// TIA Portal V17 export
// export: Created 2023-05-01T07:54:19.7526705Z, ExportSetting WithDefaults, DisplayName Totally Integrated Automation Portal, DisplayVersion V17, DisplayName TIA Portal Openness, DisplayVersion V17, DisplayName TIA Portal Version Control Interface, DisplayVersion V17, DisplayName STEP 7 Professional, DisplayVersion V17, DisplayName STEP 7 Safety, DisplayVersion V17, DisplayName WinCC Advanced / Unified PC, DisplayVersion V17
FUNCTION "FC_NormScaleAnalogInput" : Void   // FC1, LAD
{ S7_Optimized_Access := 'TRUE' }
VERSION : 0.1
// stored: AutoNumber true, IsIECCheckEnabled false, SetENOAutomatically false, UDAEnableTagReadback false
   VAR_INPUT
      AnalogInput : Int;   // Analog input [value 0 - 27648]
      minScaledValue : Real;   // lower value for scaled value Real
      maxScaledValue : Real;   // Upper value for scaled value Real
   END_VAR
   VAR_OUTPUT
      AnalogInputReal : Real;   // Scaled analog value Real
   END_VAR
   VAR_TEMP
      normAnalogValue : Real;
   END_VAR
   VAR CONSTANT
      LOWERINT : Int := 0;
      UPPERINT : Int := 27648;
   END_VAR
BEGIN

REGION Network 1
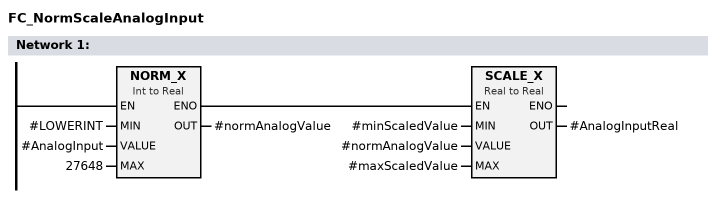
   RUNG wire#powerrail
      { S7_Templates := "[SrcType := Int, DestType := Real]" } Normalize(min := #LOWERINT, value := #AnalogInput, max := 27648, out => #normAnalogValue)
      { S7_Templates := "[SrcType := Real, DestType := Real]" } Scale(min := #minScaledValue, value := #normAnalogValue, max := #maxScaledValue, out => #AnalogInputReal)
   END_RUNG
   // the same network as SCL:
   #normAnalogValue := NORM_X(MIN := #LOWERINT, VALUE := #AnalogInput, MAX := 27648);
   #AnalogInputReal := SCALE_X(MIN := #minScaledValue, VALUE := #normAnalogValue, MAX := #maxScaledValue);
END_REGION
END_FUNCTION
